VISUALIZATION HMI_FacilityAlarm  // 2x2
END_VISUALIZATION

(* stored: Version 1.1.0.1, ProductVersion 3.1.4022.18
   Visu HMI_FacilityAlarm: Id {5dacb0d4-3ed0-447c-958f-f31a0a00a564} *)
